PROGRAM MAIN
VAR
	fbMainStateMachine			: FB_MainStateMachine;
END_VAR

fbMainStateMachine.Execute();

END_PROGRAM

(* stored: Version 1.1.0.1, ProductVersion 3.1.4024.11
   POU MAIN: Id {f3139f12-9ca1-4049-865c-64720935ee72}, SpecialFunc None *)
